PROGRAM P_UpDownSlot
VAR
	UpDownSlot_S1: FB_UpDownSlotS1;
	UpDownSlot_S2_S6: ARRAY[2..6] OF FB_UpDownSlotS2_S6;
	i:INT;
	log_ErrorEnum:UpDownSlotErrorEnum;
	log_ID:INT;


END_VAR

ACT_LOG();

//S1 急停用2904，S1-S6 只用急停按钮
(***************S1************************************************)
UpDownSlot_S1(
	timeout_up:= GVL_API.stUpDownSlot[1].timeout_up*1000, 
	timeout_down:= GVL_API.stUpDownSlot[1].timeout_down*1000, 
	extra_down_time:= GVL_API.stUpDownSlot[1].extra_down_time*1000, 
	sensor_up:= stInput.biUDS_sensor_up_S[1], 
	sensor_down:= stInput.biUDS_sensor_down_S1, 
	MoveDown_do=> , 
	MoveUp_do=>  , 
	Break=> stOutput.bqS1_Break, 
	anysensor_down=> ,
	state=> GVL_API.stUpDownSlot[1].state, 
	error_code=> GVL_API.stUpDownSlot[1].error_code, 
	error=>GVL_API.stUpDownSlot[1].Error , 
	Initialize:= GVL_API.stUpDownSlot[1].Initialize, 
	MoveDown:= GVL_API.stUpDownSlot[1].MoveDown, 
	MoveUp:= GVL_API.stUpDownSlot[1].MoveUp, 
	SetOff:= GVL_API.stUpDownSlot[1].SetOff );
	
	IF UpDownSlot_S1.MoveDown_do OR  UpDownSlot_S1.MoveUp_do THEN
		stOutput.bqS1_Drive_enabled:=TRUE;
	ELSIF NOT UpDownSlot_S1.MoveDown_do AND NOT   UpDownSlot_S1.MoveUp_do THEN 
		stOutput.bqS1_Drive_enabled:=FALSE;
	END_IF
	
	IF UpDownSlot_S1.MoveDown_do AND NOT  UpDownSlot_S1.MoveUp_do THEN 
		stOutput.bqS1_Forward_Reverse:=FALSE;
	ELSIF NOT UpDownSlot_S1.MoveDown_do AND   UpDownSlot_S1.MoveUp_do THEN 
		stOutput.bqS1_Forward_Reverse:=TRUE;
	END_IF

	GVL_API.stUpDownSlot[1].sensor_up:=stInput.biUDS_sensor_up_S[1];
	GVL_API.stUpDownSlot[1].sensor_down:=UpDownSlot_S1.anysensor_down;
	
(***************S2-S6:************************************************)
FOR i:=2 TO number_UpDownSlot DO
	UpDownSlot_S2_S6[i](
		timeout_up:=GVL_API.stUpDownSlot[i].timeout_up*1000 , 
		timeout_down:= GVL_API.stUpDownSlot[i].timeout_down*1000, 
		sensor_up:= stInput.biUDS_sensor_up_S[i], 
		MoveDown_do=> stOutput.bqUDS_MoveDown_do[i], 
		MoveUp_do=> stOutput.bqUDS_MoveUp_do[i], 
		state=> GVL_API.stUpDownSlot[i].state, 
		error_code=> GVL_API.stUpDownSlot[i].error_code, 
		error=> GVL_API.stUpDownSlot[i].Error, 
		Initialize:= GVL_API.stUpDownSlot[i].Initialize, 
		MoveDown:= GVL_API.stUpDownSlot[i].MoveDown, 
		MoveUp:= GVL_API.stUpDownSlot[i].MoveUp, 
		SetOff:=GVL_API.stUpDownSlot[i].SetOff );
		
		GVL_API.stUpDownSlot[i].sensor_up:=stInput.biUDS_sensor_up_S[i];
END_FOR

ACTION ACT_LOG:
(*************************LOG*******************************************)
log_ID:=320;
(******************s1******************************)
//initialize
AlarmActionArray[log_ID+1].AlarmMsg.EN	:='UpDownSlot1 initialize ';												
fbSetAlarm[log_ID+1](
	InUse:=TRUE , 
	EventId:=log_ID+1 , 
	EventActive:=GVL_API.stUpDownSlot[1].Initialize , 
	EventClass:=Alm_EventClass.Event , 
	ToTheLogFile:=TRUE, 
	ToTheHistory:=TRUE , 
 );
 //MoveDown
AlarmActionArray[log_ID+2].AlarmMsg.EN	:=CONCAT('UpDownSlot1 MoveDown, ',
																	LREAL_TO_STRING(GVL_API.stUpDownSlot[1].timeout_down));
AlarmActionArray[log_ID+2].AlarmMsg.EN	:=CONCAT(AlarmActionArray[log_ID+2].AlarmMsg.EN,', ');
AlarmActionArray[log_ID+2].AlarmMsg.EN	:=CONCAT(AlarmActionArray[log_ID+2].AlarmMsg.EN,
																	LREAL_TO_STRING(GVL_API.stUpDownSlot[1].extra_down_time));

fbSetAlarm[log_ID+2](
	InUse:=TRUE , 
	EventId:=log_ID+2 , 
	EventActive:=GVL_API.stUpDownSlot[1].MoveDown , 
	EventClass:=Alm_EventClass.Event , 
	ToTheLogFile:=TRUE, 
	ToTheHistory:=TRUE , 
 );
 //MoveUp
AlarmActionArray[log_ID+3].AlarmMsg.EN	:=CONCAT('UpDownSlot1 MoveUp, ',
																	LREAL_TO_STRING(GVL_API.stUpDownSlot[1].timeout_up));

fbSetAlarm[log_ID+3](
	InUse:=TRUE , 
	EventId:=log_ID+3 , 
	EventActive:=GVL_API.stUpDownSlot[1].MoveUp , 
	EventClass:=Alm_EventClass.Event , 
	ToTheLogFile:=TRUE, 
	ToTheHistory:=TRUE , 
 );

//ERROR,log_ErrorEnum只能等于一个常数
CASE GVL_API.stUpDownSlot[1].error_code  OF
0	:	log_ErrorEnum	:=	0	;
1	:	log_ErrorEnum	:=	1	;
2	:	log_ErrorEnum	:=	2	;
3	:	log_ErrorEnum	:=	3	;
4	:	log_ErrorEnum	:=	4	;
5	:	log_ErrorEnum	:=	5	;
6	:	log_ErrorEnum	:=	6	;
7	:	log_ErrorEnum	:=	7	;
666	:	log_ErrorEnum	:=	666	;

END_CASE

AlarmActionArray[log_ID+9].AlarmMsg.EN	:=CONCAT('UpDownSlot1 Error: ',TO_STRING(log_ErrorEnum));
fbSetAlarm[log_ID+9](
	InUse:=TRUE , 
	EventId:=log_ID+9 , 
	EventActive:=GVL_API.stUpDownSlot[1].error_code<>0  AND GVL_API.stUpDownSlot[1].error_code<>666, 
	EventClass:=Alm_EventClass.Alarm , 
	ToTheLogFile:=TRUE, 
	ToTheHistory:=TRUE , 
 );
 
//reset
AlarmActionArray[log_ID+10].AlarmMsg.EN	:=	'UpDownSlot1 Reset ';
fbSetAlarm[log_ID+10](
	InUse:=TRUE , 
	EventId:=log_ID+10 , 
	EventActive:=GVL_API.stUpDownSlot[1].SetOff  , 
	EventClass:=Alm_EventClass.Event , 
	ToTheLogFile:=TRUE, 
	ToTheHistory:=TRUE , 
 );
 
 
(******************s2-s6******************************)
FOR i:=2 TO number_UpDownSlot DO
//initialize
AlarmActionArray[log_ID+10*i+1].AlarmMsg.EN	:=CONCAT('UpDownSlot',
																			INT_TO_STRING(i));
AlarmActionArray[log_ID+10*i+1].AlarmMsg.EN	:=CONCAT(AlarmActionArray[log_ID+10*i+1].AlarmMsg.EN,
																			' initialize');												
fbSetAlarm[log_ID+10*i+1](
	InUse:=TRUE , 
	EventId:=log_ID+10*i+1 , 
	EventActive:=GVL_API.stUpDownSlot[i].Initialize , 
	EventClass:=Alm_EventClass.Event , 
	ToTheLogFile:=TRUE, 
	ToTheHistory:=TRUE , 
 );
 //MoveDown
 AlarmActionArray[log_ID+10*i+2].AlarmMsg.EN	:=CONCAT('UpDownSlot',
																			INT_TO_STRING(i));
AlarmActionArray[log_ID+10*i+2].AlarmMsg.EN	:=CONCAT(AlarmActionArray[log_ID+10*i+2].AlarmMsg.EN,
																			' MoveDown');
AlarmActionArray[log_ID+10*i+2].AlarmMsg.EN	:=CONCAT(AlarmActionArray[log_ID+10*i+2].AlarmMsg.EN,', ');	
AlarmActionArray[log_ID+10*i+2].AlarmMsg.EN	:=CONCAT(AlarmActionArray[log_ID+10*i+2].AlarmMsg.EN,
																	LREAL_TO_STRING(GVL_API.stUpDownSlot[i].timeout_down));

fbSetAlarm[log_ID+10*i+2](
	InUse:=TRUE , 
	EventId:=log_ID+10*i+2 , 
	EventActive:=GVL_API.stUpDownSlot[i].MoveDown , 
	EventClass:=Alm_EventClass.Event , 
	ToTheLogFile:=TRUE, 
	ToTheHistory:=TRUE , 
 );
 //MoveUp
AlarmActionArray[log_ID+10*i+3].AlarmMsg.EN	:=CONCAT('UpDownSlot',
																			INT_TO_STRING(i));
AlarmActionArray[log_ID+10*i+3].AlarmMsg.EN	:=CONCAT(AlarmActionArray[log_ID+10*i+3].AlarmMsg.EN,
																			' MoveUp');
AlarmActionArray[log_ID+10*i+3].AlarmMsg.EN	:=CONCAT(AlarmActionArray[log_ID+10*i+3].AlarmMsg.EN,', ');	
AlarmActionArray[log_ID+10*i+3].AlarmMsg.EN	:=CONCAT(AlarmActionArray[log_ID+10*i+3].AlarmMsg.EN,
																	LREAL_TO_STRING(GVL_API.stUpDownSlot[i].timeout_up));

fbSetAlarm[log_ID+10*i+3](
	InUse:=TRUE , 
	EventId:=log_ID+10*i+3 , 
	EventActive:=GVL_API.stUpDownSlot[i].MoveUp , 
	EventClass:=Alm_EventClass.Event , 
	ToTheLogFile:=TRUE, 
	ToTheHistory:=TRUE , 
 );

//ERROR,log_ErrorEnum只能等于一个常数
CASE GVL_API.stUpDownSlot[i].error_code  OF
0	:	log_ErrorEnum	:=	0	;
1	:	log_ErrorEnum	:=	1	;
2	:	log_ErrorEnum	:=	2	;
3	:	log_ErrorEnum	:=	3	;
4	:	log_ErrorEnum	:=	4	;
5	:	log_ErrorEnum	:=	5	;
6	:	log_ErrorEnum	:=	6	;
7	:	log_ErrorEnum	:=	7	;
666	:	log_ErrorEnum	:=	666	;


END_CASE
AlarmActionArray[log_ID+10*i+9].AlarmMsg.EN	:=CONCAT('UpDownSlot',INT_TO_STRING(i));
AlarmActionArray[log_ID+10*i+9].AlarmMsg.EN	:=CONCAT(AlarmActionArray[log_ID+10*i+9].AlarmMsg.EN,
																			' Error: ');
AlarmActionArray[log_ID+10*i+9].AlarmMsg.EN	:=CONCAT(AlarmActionArray[log_ID+10*i+9].AlarmMsg.EN,
																			TO_STRING(log_ErrorEnum));																			

fbSetAlarm[log_ID+10*i+9](
	InUse:=TRUE , 
	EventId:=log_ID+10*i+9 , 
	EventActive:=GVL_API.stUpDownSlot[i].error_code<>0 AND GVL_API.stUpDownSlot[i].error_code<>666 , 
	EventClass:=Alm_EventClass.Alarm , 
	ToTheLogFile:=TRUE, 
	ToTheHistory:=TRUE , 
 );
 
//reset
AlarmActionArray[log_ID+10*i+10].AlarmMsg.EN	:=CONCAT('UpDownSlot',
																			INT_TO_STRING(i));
AlarmActionArray[log_ID+10*i+10].AlarmMsg.EN	:=CONCAT(AlarmActionArray[log_ID+10*i+10].AlarmMsg.EN,
																			' Reset');		

fbSetAlarm[log_ID+10*i+10](
	InUse:=TRUE , 
	EventId:=log_ID+10*i+10 , 
	EventActive:=GVL_API.stUpDownSlot[i].SetOff  , 
	EventClass:=Alm_EventClass.Event , 
	ToTheLogFile:=TRUE, 
	ToTheHistory:=TRUE , 
 );
END_FOR
 (*************em-stop*     *************
 AlarmActionArray[399].AlarmMsg.EN	:='UpDownSlot Error: emergency_error';																		

fbSetAlarm[399](
	InUse:=TRUE , 
	EventId:=399 , 
	EventActive:=GVL_API.stUpDownSlot[i].error_code=666 , 
	EventClass:=Alm_EventClass.Alarm , 
	ToTheLogFile:=TRUE, 
	ToTheHistory:=TRUE , 
 );
*)
END_ACTION

END_PROGRAM

(* stored: Version 1.1.0.1, ProductVersion 3.1.4024.11
   POU P_UpDownSlot: Id {1e93bc92-b601-49b4-8de9-efab48533a3d}, SpecialFunc None
   Action ACT_LOG: Id {cf8c18b0-2a56-4fa5-a3af-c22ce0ab5f69} *)
